// TIA Portal V17 export
// export: Created 2024-09-02T12:50:17.1770288Z, ExportSetting WithDefaults, DisplayName Totally Integrated Automation Portal, DisplayVersion V17, DisplayName TIA Portal Openness, DisplayVersion V17, DisplayName TIA Portal Version Control Interface, DisplayVersion V17, DisplayName STEP 7 Professional, DisplayVersion V17, DisplayName STEP 7 Safety, DisplayVersion V17, DisplayName WinCC Professional, DisplayVersion V17
DATA_BLOCK "SysDB_MP_Function_OP70"   // DB254
{ S7_Optimized_Access := 'TRUE'; DB_Accessible_From_OPC_UA := 'FALSE' }
AUTHOR : OlegFuehrus
FAMILY : BA
NAME : BA
VERSION : 0.1
// stored: AutoNumber true, DBAccessibleFromOPCUA false, IsOnlyStoredInLoadMemory false, IsRetainMemResEnabled false, IsWriteProtectedInAS false, MemoryReserve 100
   VAR
      Deselection_aktiv { ExternalWritable := 'False'} : Bool;
      Setup { S7_SetPoint := 'True'} : "TypeFunction";
      PowerUp { S7_SetPoint := 'True'} : "TypeFunction";
      Unit { S7_SetPoint := 'True'} : "TypeFunction";
      NutRunner { S7_SetPoint := 'True'} : "TypeFunction";
      NutRunnerGroup { S7_SetPoint := 'True'} : "TypeFunction";
      CycleType { S7_SetPoint := 'True'} : "TypeFunction";
      UserDefine { S7_SetPoint := 'True'} : "TypeFunction";
   END_VAR
BEGIN
END_DATA_BLOCK
